// TIA Portal V19 export
TYPE "C701_VAR_IF_VEB_TYPIC"
   STRUCT
      REQ_VE { ExternalAccessible := 'False'; ExternalVisible := 'False'; ExternalWritable := 'False'} : Bool;   // Warmtevraag voor kring verwarmingsbatterijen
      STO { ExternalAccessible := 'False'; ExternalVisible := 'False'; ExternalWritable := 'False'} : Struct   // Opsomming van alle storingen
         A001 : Bool;   // Ruimtetemperatuur te laag
         A002 : Bool;   // Fout temperatuurmeting
      END_STRUCT;
   END_STRUCT;
END_TYPE
